{attribute 'linkalways'}
{attribute 'no_explicit_call' := 'This FB is a CLASS and must be accessed using methods or properties'}
{attribute 'enable_dynamic_creation'}
FUNCTION_BLOCK Node_F_VN_ConvertPolarToCartesianImages EXTENDS VisionNode
VAR
    ipSrcImageMag : _ITcVnImage;
    ipSrcImageAng : _ITcVnImage;
    ipDestImageX : _ITcVnImage;
    ipDestImageY : _ITcVnImage;
    hrPrev : _HRESULT(S_OK);
    hresult : _HRESULT(S_OK);
END_VAR

METHOD PUBLIC Clone : I_Node
VAR
    pNode : POINTER TO Node_F_VN_ConvertPolarToCartesianImages;
END_VAR
pNode := __NEW(Node_F_VN_ConvertPolarToCartesianImages);
Clone := pNode^;
END_METHOD

METHOD FB_init : BOOL
VAR_INPUT
    bInitRetains : BOOL;
    bInCopyCode : BOOL;
END_VAR
AddInput('ipSrcImageMag', ipSrcImageMag);
AddInput('ipSrcImageAng', ipSrcImageAng);
AddOutput('ipDestImageX', ipDestImageX);
AddOutput('ipDestImageY', ipDestImageY);
AddInput('hrPrev', hrPrev);
AddOutput('hresult', hresult);
END_METHOD

METHOD PROTECTED OnExecute
hresult.Value := F_VN_ConvertPolarToCartesianImages(
    ipSrcImageMag := ipSrcImageMag.Value,
    ipSrcImageAng := ipSrcImageAng.Value,
    ipDestImageX := ipDestImageX.Value,
    ipDestImageY := ipDestImageY.Value,
    hrPrev := hrPrev.Value);
END_METHOD

METHOD PUBLIC PreExecutionCheck
VAR_INPUT
    Check : I_PreExecutionChecks;
END_VAR
Check.IsTrue(ipSrcImageMag.IsValid, 'ipSrcImageMag must contain an image');
Check.IsTrue(ipSrcImageMag.IsElementType(ETcVnElementType.TCVN_ET_REAL) OR
             ipSrcImageMag.IsElementType(ETcVnElementType.TCVN_ET_LREAL), 'Coordinate images must contain REAL or LREAL elements');
Check.IsTrue(ipSrcImageAng.IsValid, 'ipSrcImageAng must contain an image');
Check.IsTrue(ImagesHaveMatchingPixelFormats(ipSrcImageMag.Value, ipSrcImageAng.Value), 'Source images must have matching pixel formats');
Check.IsTrue(IsImage1SizeEqualToImage2Size(ipSrcImageMag.Value, ipSrcImageAng.Value), 'Source images must have matching dimensions');
END_METHOD

END_FUNCTION_BLOCK

(* stored: Version 1.1.0.1, ProductVersion 3.1.4026.19
   POU Node_F_VN_ConvertPolarToCartesianImages: Id {82ac119b-765e-47bd-ba7e-e1a89fdcafdd}, SpecialFunc None
   Folder Constructor: Id {cdc5f6d4-1f64-073d-0785-62509f541e00}
   Method Clone: Id {db04050f-ecc8-4c83-9cb6-ce099336a463}
   Method FB_init: Id {e90c0ac6-0bba-4f49-a41d-17fc7338c3ae}
   Method OnExecute: Id {29cae259-6d6c-4ba8-ad6b-7cea51aa0f32}
   Method PreExecutionCheck: Id {23da948d-d5d7-4923-ab85-03ac41049353} *)
